// TIA Portal V21 export
FUNCTION "GestPid_Comando2Motori" : Void   // FC64, LAD
{ S7_Optimized_Access := 'TRUE' }
// stored: SetENOAutomatically false
   VAR_INPUT
      K_Motore1 : Int;
      K_Motore2 : Int;
      K_Pid : Int;
   END_VAR
BEGIN

REGION Network 1 (SCL)
   "Pid".P[#K_Pid].In.K_Motore1 := #K_Motore1;
   "Pid".P[#K_Pid].In.K_Motore2 := #K_Motore2;
END_REGION
END_FUNCTION
